(* Logix 5000 project; controller p65 vendor 1 type 14 code 85 rev 20.11; software revision 20.01; part 7 of 7 *)
(* tags used below, declared in another part *)
   Commpower : ALIAS FOR REAL00_102;
   DCMicroGridisSimulating : ALIAS FOR DINT00_23.10;
   House01current : ALIAS FOR REAL00_117;
   House01isConnected : ALIAS FOR DINT00_28.23;
   House02current : ALIAS FOR REAL00_130;
   House02isConnected : ALIAS FOR DINT00_29.13;
   House03current : ALIAS FOR REAL00_143;
   House03isConnected : ALIAS FOR DINT00_30.3;
   House04current : ALIAS FOR REAL00_156;
   House04isConnected : ALIAS FOR DINT00_30.25;
   House05current : ALIAS FOR REAL00_169;
   House05isConnected : ALIAS FOR DINT00_31.15;
   LastSolar_Power : REAL;
   Load01isConnected : ALIAS FOR DINT00_24.13;
   Load02isConnected : ALIAS FOR DINT00_25.3;
   Load03isConnected : ALIAS FOR DINT00_25.25;
   Load04isConnected : ALIAS FOR DINT00_26.15;
   Load05isConnected : ALIAS FOR DINT00_27.5;
   Loadsaccum : ALIAS FOR REAL00_30;
   Loadscurrent : ALIAS FOR REAL00_105;
   LoadscurrentHILS : ALIAS FOR plc1_local_5[0];
   LoadscurrentRaw : ALIAS FOR Local:1:I.Ch6Data;
   Loadsdifference : ALIAS FOR REAL00_106;
   LoadslastLowVoltage : ALIAS FOR DINT00_27.22;
   LoadslowVoltage : ALIAS FOR DINT00_27.23;
   LoadslowVoltageBound : ALIAS FOR REAL00_107;
   Loadspower : ALIAS FOR REAL00_108;
   Loadsrecovered : ALIAS FOR DINT00_27.24;
   LoadssampleNow : ALIAS FOR DINT00_32.3;
   LoadssampleTimer : ALIAS FOR CLTIMER00_89;
   Loadstotal : ALIAS FOR REAL00_183;
   LoadstotalTooLarge : ALIAS FOR DINT00_32.4;
   LoadstotalTooSmall : ALIAS FOR DINT00_32.5;
   Loadsvoltage : ALIAS FOR REAL00_184;
   LoadsVoltageBalanceEventFail : ALIAS FOR DINT00_32.6;
   LoadsVoltageBalanceEventSuccess : ALIAS FOR DINT00_32.7;
   LoadsVoltageBalanceFailTimer : ALIAS FOR CLTIMER00_90;
   LoadsVoltageBalanceInProcess : ALIAS FOR DINT00_32.8;
   LoadsVoltageBalanceMsg : ALIAS FOR MESSAGE00_23;
   LoadsVoltageBalanceSuccessTimer : ALIAS FOR CLTIMER00_91;
   LoadsvoltageHILS : ALIAS FOR plc1_local_5[1];
   LoadsvoltageRaw : ALIAS FOR Local:1:I.Ch8Data;
   LoadsVoltageRebalancedEventFail : ALIAS FOR DINT00_32.9;
   LoadsVoltageRebalancedEventSuccess : ALIAS FOR DINT00_32.10;
   LoadsVoltageRebalancedFailTimer : ALIAS FOR CLTIMER00_92;
   LoadsVoltageRebalancedInProcess : ALIAS FOR DINT00_32.11;
   LoadsVoltageRebalancedMsg : ALIAS FOR MESSAGE00_24;
   LoadsVoltageRebalancedSuccessTimer : ALIAS FOR CLTIMER00_93;
   Resaccum : ALIAS FOR REAL00_109;
   ResBattempt : ALIAS FOR DINT00_10;
   ResBclose : ALIAS FOR Local:3:O.Data.10;
   ResBcloseHILS : ALIAS FOR plc1_local_6[0].10;
   ResBcloseProxy : ALIAS FOR DINT00_27.25;
   ResBdeadBand : ALIAS FOR REAL00_110;
   ResBfailedToOpen : ALIAS FOR DINT00_27.26;
   ResBintForceOpen : ALIAS FOR DINT00_27.27;
   ResBintReqClose : ALIAS FOR DINT00_27.28;
   ResBisClosed : ALIAS FOR DINT00_27.29;
   ResBisOpen : ALIAS FOR DINT00_27.30;
   ResBmaxAttempts : ALIAS FOR DINT00_11;
   ResBmaxLoadCurrent : ALIAS FOR REAL00_111;
   ResBopenTimer : ALIAS FOR CLTIMER00_48;
   ResBreqClose : ALIAS FOR DINT00_27.31;
   ResBreqOpen : ALIAS FOR DINT00_28.0;
   ResBreqReset : ALIAS FOR DINT00_28.1;
   ResBretriesFailed : ALIAS FOR DINT00_28.2;
   ResBtooMuchCurrent : ALIAS FOR DINT00_28.3;
   ResBunexpectedLowCurrent : ALIAS FOR DINT00_28.4;
   RescanNotifyUser : ALIAS FOR DINT00_28.5;
   RescommandChanged : ALIAS FOR DINT00_28.6;
   RescommandChangedTimer : ALIAS FOR CLTIMER00_49;
   Rescurrent : ALIAS FOR REAL00_112;
   RescurrentHILS : ALIAS FOR plc1_local_3[6];
   RescurrentRaw : ALIAS FOR Local:1:I.Ch11Data;
   Resdeadband : ALIAS FOR REAL00_113;
   Resdifference : ALIAS FOR REAL00_114;
   ResfailedToConnect : ALIAS FOR DINT00_28.7;
   ResfailedToDisconnect : ALIAS FOR DINT00_28.8;
   ResintReqConnect : ALIAS FOR DINT00_31.23;
   ResisConnected : ALIAS FOR DINT00_31.24;
   ResisDisconnected : ALIAS FOR DINT00_31.25;
   ResnotificationTimer : ALIAS FOR CLTIMER00_85;
   ResOverCurrentConditionEventFail : ALIAS FOR DINT00_31.26;
   ResOverCurrentConditionEventSuccess : ALIAS FOR DINT00_31.27;
   ResOverCurrentConditionFailTimer : ALIAS FOR CLTIMER00_86;
   ResOverCurrentConditionInProcess : ALIAS FOR DINT00_31.28;
   ResOverCurrentConditionMsg : ALIAS FOR MESSAGE00_22;
   ResOverCurrentConditionSuccessTimer : ALIAS FOR CLTIMER00_87;
   Respower : ALIAS FOR REAL00_180;
   ResreqConnect : ALIAS FOR DINT00_31.29;
   ResreqDisconnect : ALIAS FOR DINT00_31.30;
   RessampleNow : ALIAS FOR DINT00_31.31;
   RessampleTimer : ALIAS FOR CLTIMER00_88;
   Restotal : ALIAS FOR REAL00_181;
   RestotalTooLarge : ALIAS FOR DINT00_32.0;
   RestotalTooSmall : ALIAS FOR DINT00_32.1;
   ResuserNotified : ALIAS FOR DINT00_32.2;
   Resvoltage : ALIAS FOR REAL00_182;
   ResvoltageHILS : ALIAS FOR plc1_local_3[7];
   ResvoltageRaw : ALIAS FOR Local:2:I.Ch1Data;
   Solar_Power : ALIAS FOR plc1_local_1[0];
   SolarMeasureTimer : TIMER;
   SolarPanelBclose : ALIAS FOR Local:3:O.Data.13;
   SolarPanelBcloseHILS : ALIAS FOR plc1_local_6[0].12;
   SolarPanelBcloseProxy : ALIAS FOR DINT00_32.22;
   SolarPanelBintReqClose : ALIAS FOR DINT00_32.23;
   SolarPanelBisClosed : ALIAS FOR DINT00_32.24;
   SolarPanelBisOpen : ALIAS FOR DINT00_32.25;
   SolarPanelBreqClose : ALIAS FOR DINT00_32.26;
   SolarPanelBreqOpen : ALIAS FOR DINT00_32.27;
   SolarPanelcanSupplyPower : ALIAS FOR DINT00_32.28;
   SolarPanelcommandChanged : ALIAS FOR DINT00_32.29;
   SolarPanelcommandChangedTimer : ALIAS FOR CLTIMER00_99;
   SolarPanelcurrent : ALIAS FOR REAL00_187;
   SolarPanelcurrentHILS : ALIAS FOR plc1_local_3[0];
   SolarPanelcurrentRaw : ALIAS FOR Local:1:I.Ch2Data;
   SolarPaneldeadband : ALIAS FOR REAL00_188;
   SolarPanelfailedToConnect : ALIAS FOR DINT00_32.30;
   SolarPanelfailedToDisconnect : ALIAS FOR DINT00_32.31;
   SolarPanelintReqConnect : ALIAS FOR DINT00_33.0;
   SolarPanelisConnected : ALIAS FOR DINT00_33.1;
   SolarPanelisDisconnected : ALIAS FOR DINT00_33.2;
   SolarPanelisFunctional : ALIAS FOR DINT00_33.3;
   SolarPanelpower : ALIAS FOR REAL00_190;
   SolarPanelprovidingExcessPower : ALIAS FOR DINT00_33.4;
   SolarPanelreqConnect : ALIAS FOR DINT00_33.5;
   SolarPanelreqDisconnect : ALIAS FOR DINT00_33.6;
   SolarPanelvoltage : ALIAS FOR REAL00_191;
   SolarPanelvoltageHILS : ALIAS FOR plc1_local_3[1];
   SolarPanelvoltageRaw : ALIAS FOR Local:1:I.Ch1Data;
   UsingAgents : BOOL;

PROGRAM Loads   (* main routine Loads *)
VAR
   VoltageRebalancePhase : DINT;
END_VAR

ROUTINE Loads   (* ladder *)
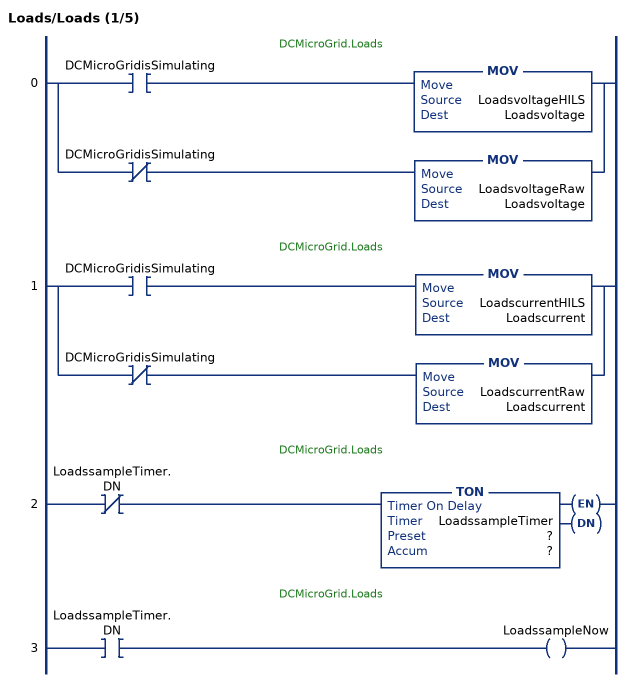
   // DCMicroGrid.Loads
   0: [XIC(DCMicroGridisSimulating) MOV(LoadsvoltageHILS,Loadsvoltage) ,XIO(DCMicroGridisSimulating) MOV(LoadsvoltageRaw,Loadsvoltage) ];
   // DCMicroGrid.Loads
   1: [XIC(DCMicroGridisSimulating) MOV(LoadscurrentHILS,Loadscurrent) ,XIO(DCMicroGridisSimulating) MOV(LoadscurrentRaw,Loadscurrent) ];
   // DCMicroGrid.Loads
   2: XIO(LoadssampleTimer.DN)TON(LoadssampleTimer,?,?);
   // DCMicroGrid.Loads
   3: XIC(LoadssampleTimer.DN)OTE(LoadssampleNow);
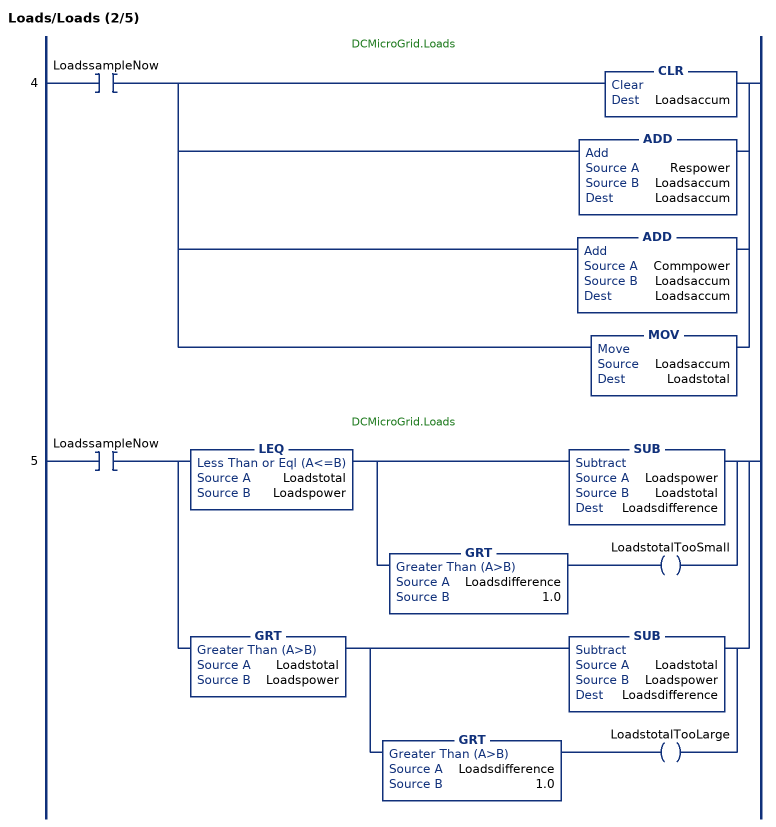
   // DCMicroGrid.Loads
   4: XIC(LoadssampleNow)[CLR(Loadsaccum) ,[ADD(Respower,Loadsaccum,Loadsaccum) ,ADD(Commpower,Loadsaccum,Loadsaccum) ] ,MOV(Loadsaccum,Loadstotal) ];
   // DCMicroGrid.Loads
   5: XIC(LoadssampleNow)[LEQ(Loadstotal,Loadspower) [SUB(Loadspower,Loadstotal,Loadsdifference) ,GRT(Loadsdifference,1.0) OTE(LoadstotalTooSmall) ] ,GRT(Loadstotal,Loadspower) [SUB(Loadstotal,Loadspower,Loadsdifference) ,GRT(Loadsdifference,1.0) OTE(LoadstotalTooLarge) ] ];
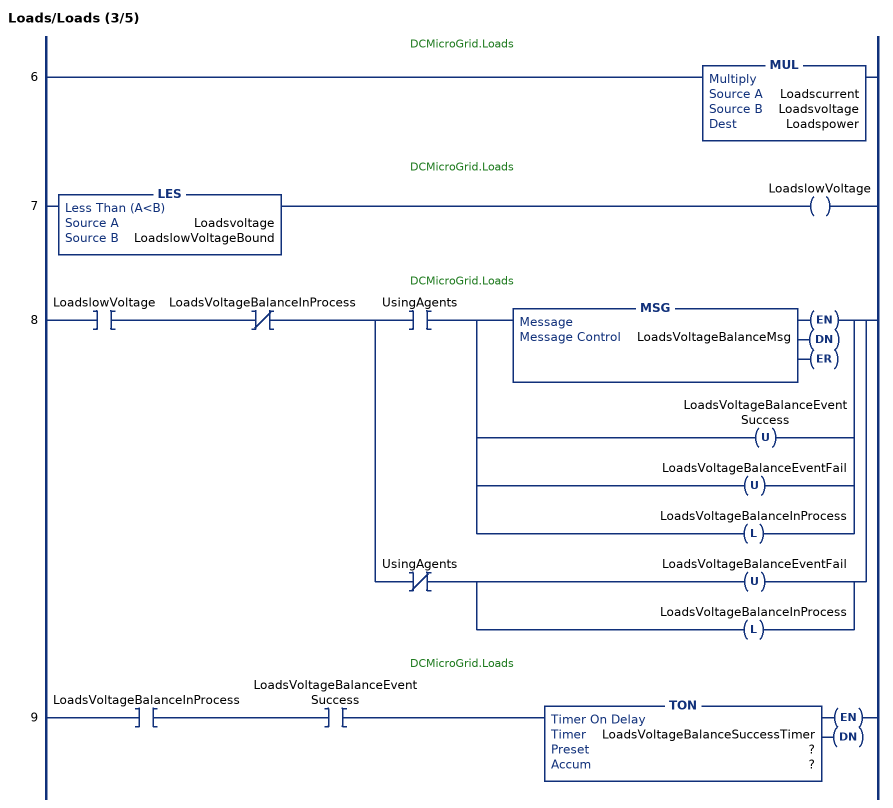
   // DCMicroGrid.Loads
   6: MUL(Loadscurrent,Loadsvoltage,Loadspower);
   // DCMicroGrid.Loads
   7: LES(Loadsvoltage,LoadslowVoltageBound)OTE(LoadslowVoltage);
   // DCMicroGrid.Loads
   8: XIC(LoadslowVoltage)XIO(LoadsVoltageBalanceInProcess)[XIC(UsingAgents) [MSG(LoadsVoltageBalanceMsg) ,OTU(LoadsVoltageBalanceEventSuccess) ,OTU(LoadsVoltageBalanceEventFail) ,OTL(LoadsVoltageBalanceInProcess) ] ,XIO(UsingAgents) [OTU(LoadsVoltageBalanceEventFail) ,OTL(LoadsVoltageBalanceInProcess) ] ];
   // DCMicroGrid.Loads
   9: XIC(LoadsVoltageBalanceInProcess)XIC(LoadsVoltageBalanceEventSuccess)TON(LoadsVoltageBalanceSuccessTimer,?,?);
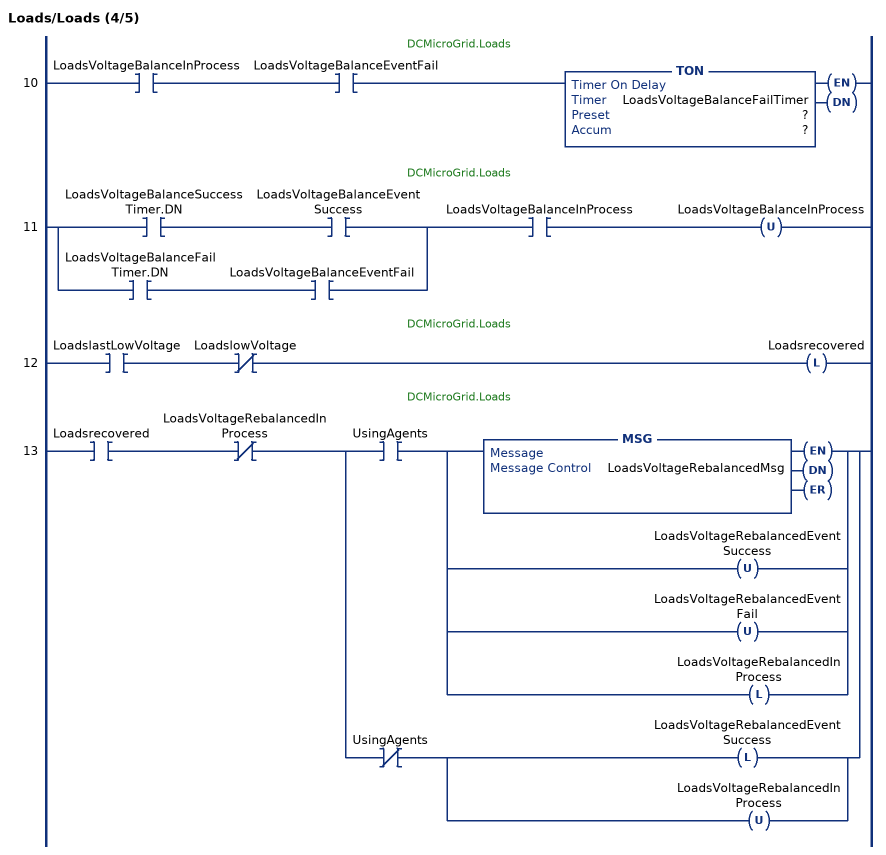
   // DCMicroGrid.Loads
   10: XIC(LoadsVoltageBalanceInProcess)XIC(LoadsVoltageBalanceEventFail)TON(LoadsVoltageBalanceFailTimer,?,?);
   // DCMicroGrid.Loads
   11: [XIC(LoadsVoltageBalanceSuccessTimer.DN) XIC(LoadsVoltageBalanceEventSuccess) ,XIC(LoadsVoltageBalanceFailTimer.DN) XIC(LoadsVoltageBalanceEventFail) ]XIC(LoadsVoltageBalanceInProcess)OTU(LoadsVoltageBalanceInProcess);
   // DCMicroGrid.Loads
   12: XIC(LoadslastLowVoltage)XIO(LoadslowVoltage)OTL(Loadsrecovered);
   // DCMicroGrid.Loads
   13: XIC(Loadsrecovered)XIO(LoadsVoltageRebalancedInProcess)[XIC(UsingAgents) [MSG(LoadsVoltageRebalancedMsg) ,OTU(LoadsVoltageRebalancedEventSuccess) ,OTU(LoadsVoltageRebalancedEventFail) ,OTL(LoadsVoltageRebalancedInProcess) ] ,XIO(UsingAgents) [OTL(LoadsVoltageRebalancedEventSuccess) ,OTU(LoadsVoltageRebalancedInProcess) ] ];
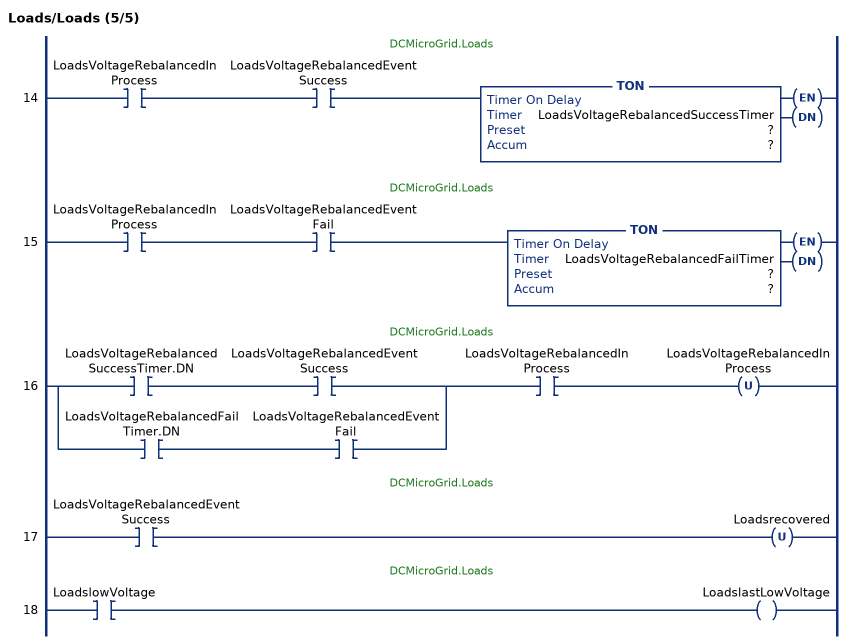
   // DCMicroGrid.Loads
   14: XIC(LoadsVoltageRebalancedInProcess)XIC(LoadsVoltageRebalancedEventSuccess)TON(LoadsVoltageRebalancedSuccessTimer,?,?);
   // DCMicroGrid.Loads
   15: XIC(LoadsVoltageRebalancedInProcess)XIC(LoadsVoltageRebalancedEventFail)TON(LoadsVoltageRebalancedFailTimer,?,?);
   // DCMicroGrid.Loads
   16: [XIC(LoadsVoltageRebalancedSuccessTimer.DN) XIC(LoadsVoltageRebalancedEventSuccess) ,XIC(LoadsVoltageRebalancedFailTimer.DN) XIC(LoadsVoltageRebalancedEventFail) ]XIC(LoadsVoltageRebalancedInProcess)OTU(LoadsVoltageRebalancedInProcess);
   // DCMicroGrid.Loads
   17: XIC(LoadsVoltageRebalancedEventSuccess)OTU(Loadsrecovered);
   // DCMicroGrid.Loads
   18: XIC(LoadslowVoltage)OTE(LoadslastLowVoltage);
END_ROUTINE
END_PROGRAM

PROGRAM Main   (* main routine PDLGeneratedControlLogic *)

ROUTINE PDLGeneratedControlLogic   (* ladder *)
END_ROUTINE
END_PROGRAM

PROGRAM Res   (* main routine Res *)

ROUTINE Res   (* ladder *)
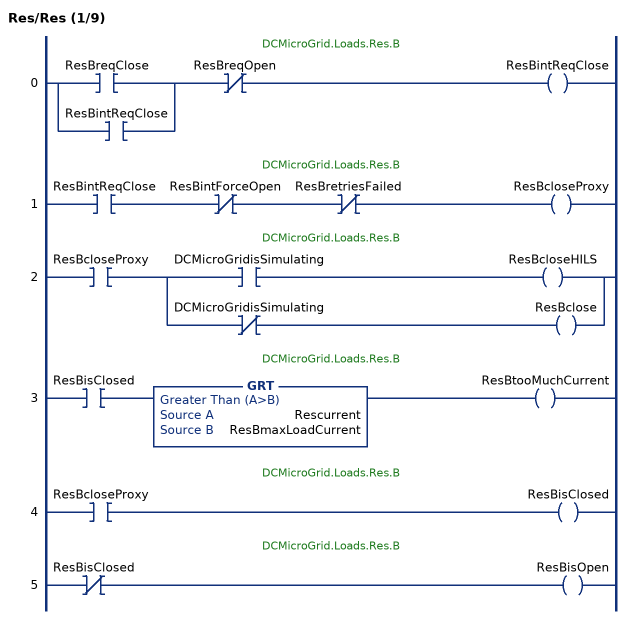
   // DCMicroGrid.Loads.Res.B
   0: [XIC(ResBreqClose) ,XIC(ResBintReqClose) ]XIO(ResBreqOpen)OTE(ResBintReqClose);
   // DCMicroGrid.Loads.Res.B
   1: XIC(ResBintReqClose)XIO(ResBintForceOpen)XIO(ResBretriesFailed)OTE(ResBcloseProxy);
   // DCMicroGrid.Loads.Res.B
   2: XIC(ResBcloseProxy)[XIC(DCMicroGridisSimulating) OTE(ResBcloseHILS) ,XIO(DCMicroGridisSimulating) OTE(ResBclose) ];
   // DCMicroGrid.Loads.Res.B
   3: XIC(ResBisClosed)GRT(Rescurrent,ResBmaxLoadCurrent)OTE(ResBtooMuchCurrent);
   // DCMicroGrid.Loads.Res.B
   4: XIC(ResBcloseProxy)OTE(ResBisClosed);
   // DCMicroGrid.Loads.Res.B
   5: XIO(ResBisClosed)OTE(ResBisOpen);
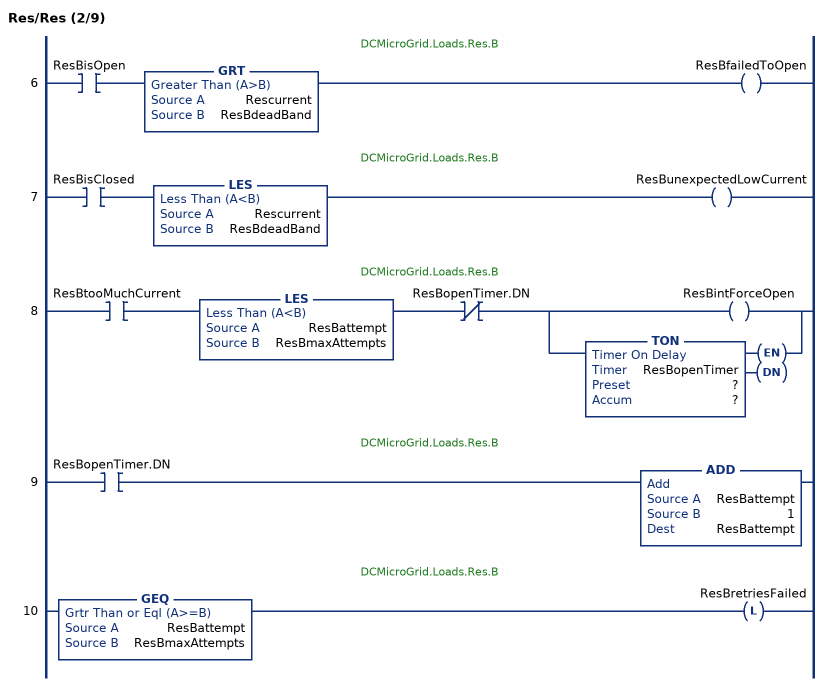
   // DCMicroGrid.Loads.Res.B
   6: XIC(ResBisOpen)GRT(Rescurrent,ResBdeadBand)OTE(ResBfailedToOpen);
   // DCMicroGrid.Loads.Res.B
   7: XIC(ResBisClosed)LES(Rescurrent,ResBdeadBand)OTE(ResBunexpectedLowCurrent);
   // DCMicroGrid.Loads.Res.B
   8: XIC(ResBtooMuchCurrent)LES(ResBattempt,ResBmaxAttempts)XIO(ResBopenTimer.DN)[OTE(ResBintForceOpen) ,TON(ResBopenTimer,?,?) ];
   // DCMicroGrid.Loads.Res.B
   9: XIC(ResBopenTimer.DN)ADD(ResBattempt,1,ResBattempt);
   // DCMicroGrid.Loads.Res.B
   10: GEQ(ResBattempt,ResBmaxAttempts)OTL(ResBretriesFailed);
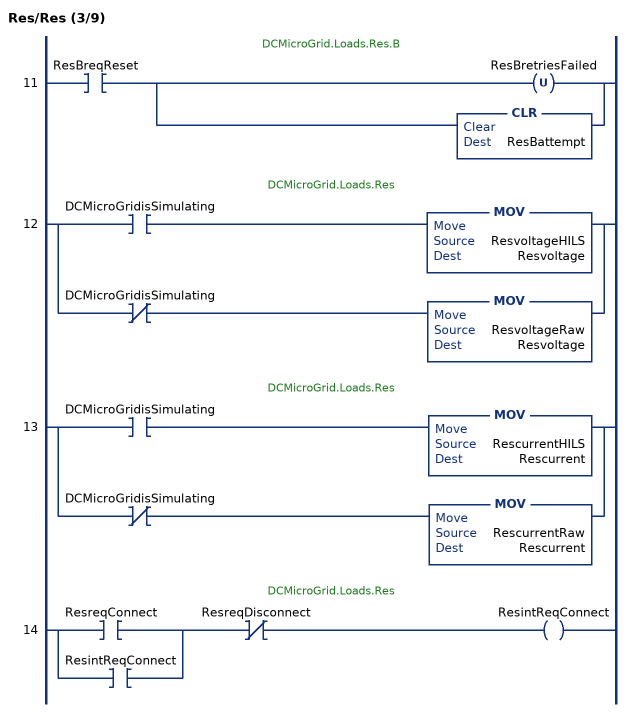
   // DCMicroGrid.Loads.Res.B
   11: XIC(ResBreqReset)[OTU(ResBretriesFailed) ,CLR(ResBattempt) ];
   // DCMicroGrid.Loads.Res
   12: [XIC(DCMicroGridisSimulating) MOV(ResvoltageHILS,Resvoltage) ,XIO(DCMicroGridisSimulating) MOV(ResvoltageRaw,Resvoltage) ];
   // DCMicroGrid.Loads.Res
   13: [XIC(DCMicroGridisSimulating) MOV(RescurrentHILS,Rescurrent) ,XIO(DCMicroGridisSimulating) MOV(RescurrentRaw,Rescurrent) ];
   // DCMicroGrid.Loads.Res
   14: [XIC(ResreqConnect) ,XIC(ResintReqConnect) ]XIO(ResreqDisconnect)OTE(ResintReqConnect);
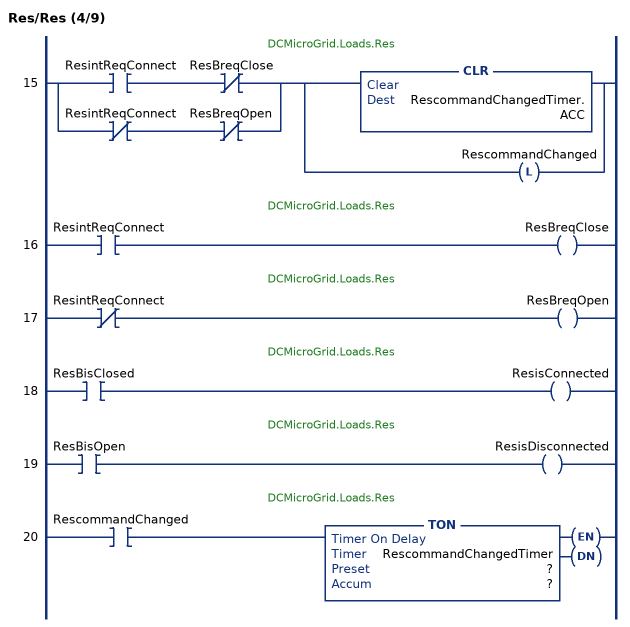
   // DCMicroGrid.Loads.Res
   15: [XIC(ResintReqConnect) XIO(ResBreqClose) ,XIO(ResintReqConnect) XIO(ResBreqOpen) ][CLR(RescommandChangedTimer.ACC) ,OTL(RescommandChanged) ];
   // DCMicroGrid.Loads.Res
   16: XIC(ResintReqConnect)OTE(ResBreqClose);
   // DCMicroGrid.Loads.Res
   17: XIO(ResintReqConnect)OTE(ResBreqOpen);
   // DCMicroGrid.Loads.Res
   18: XIC(ResBisClosed)OTE(ResisConnected);
   // DCMicroGrid.Loads.Res
   19: XIC(ResBisOpen)OTE(ResisDisconnected);
   // DCMicroGrid.Loads.Res
   20: XIC(RescommandChanged)TON(RescommandChangedTimer,?,?);
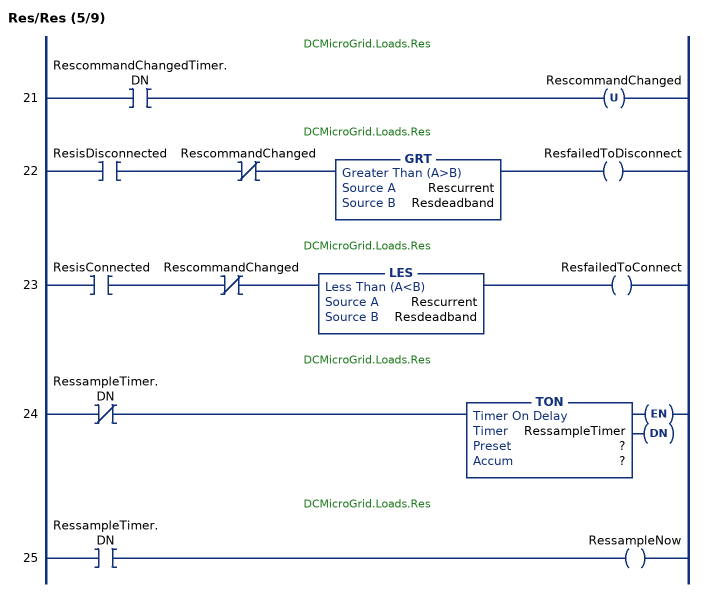
   // DCMicroGrid.Loads.Res
   21: XIC(RescommandChangedTimer.DN)OTU(RescommandChanged);
   // DCMicroGrid.Loads.Res
   22: XIC(ResisDisconnected)XIO(RescommandChanged)GRT(Rescurrent,Resdeadband)OTE(ResfailedToDisconnect);
   // DCMicroGrid.Loads.Res
   23: XIC(ResisConnected)XIO(RescommandChanged)LES(Rescurrent,Resdeadband)OTE(ResfailedToConnect);
   // DCMicroGrid.Loads.Res
   24: XIO(RessampleTimer.DN)TON(RessampleTimer,?,?);
   // DCMicroGrid.Loads.Res
   25: XIC(RessampleTimer.DN)OTE(RessampleNow);
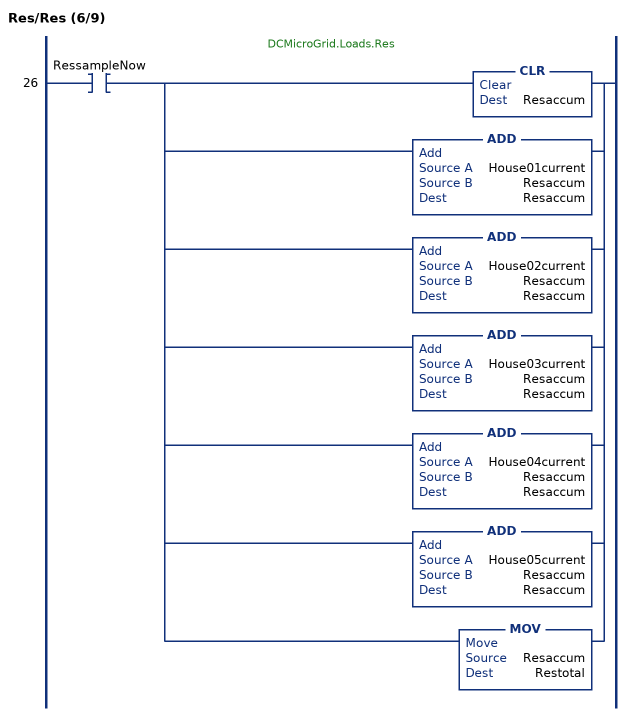
   // DCMicroGrid.Loads.Res
   26: XIC(RessampleNow)[CLR(Resaccum) ,[ADD(House01current,Resaccum,Resaccum) ,ADD(House02current,Resaccum,Resaccum) ,ADD(House03current,Resaccum,Resaccum) ,ADD(House04current,Resaccum,Resaccum) ,ADD(House05current,Resaccum,Resaccum) ] ,MOV(Resaccum,Restotal) ];
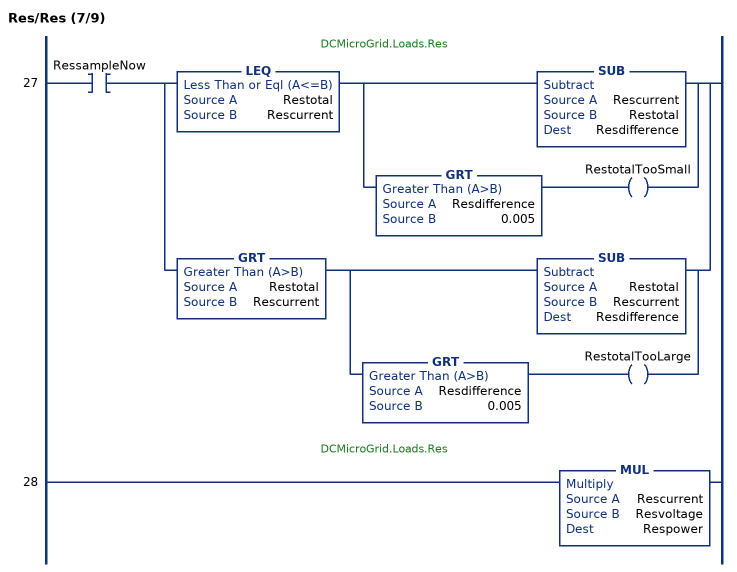
   // DCMicroGrid.Loads.Res
   27: XIC(RessampleNow)[LEQ(Restotal,Rescurrent) [SUB(Rescurrent,Restotal,Resdifference) ,GRT(Resdifference,0.005) OTE(RestotalTooSmall) ] ,GRT(Restotal,Rescurrent) [SUB(Restotal,Rescurrent,Resdifference) ,GRT(Resdifference,0.005) OTE(RestotalTooLarge) ] ];
   // DCMicroGrid.Loads.Res
   28: MUL(Rescurrent,Resvoltage,Respower);
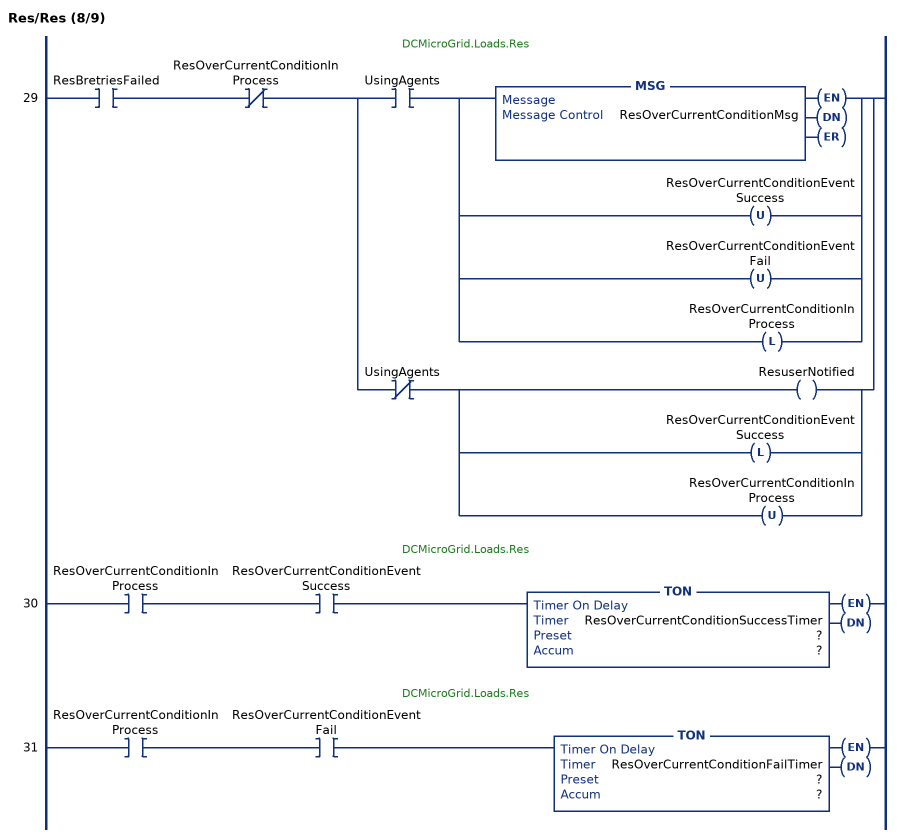
   // DCMicroGrid.Loads.Res
   29: XIC(ResBretriesFailed)XIO(ResOverCurrentConditionInProcess)[XIC(UsingAgents) [MSG(ResOverCurrentConditionMsg) ,OTU(ResOverCurrentConditionEventSuccess) ,OTU(ResOverCurrentConditionEventFail) ,OTL(ResOverCurrentConditionInProcess) ] ,XIO(UsingAgents) [OTE(ResuserNotified) ,OTL(ResOverCurrentConditionEventSuccess) ,OTU(ResOverCurrentConditionInProcess) ] ];
   // DCMicroGrid.Loads.Res
   30: XIC(ResOverCurrentConditionInProcess)XIC(ResOverCurrentConditionEventSuccess)TON(ResOverCurrentConditionSuccessTimer,?,?);
   // DCMicroGrid.Loads.Res
   31: XIC(ResOverCurrentConditionInProcess)XIC(ResOverCurrentConditionEventFail)TON(ResOverCurrentConditionFailTimer,?,?);
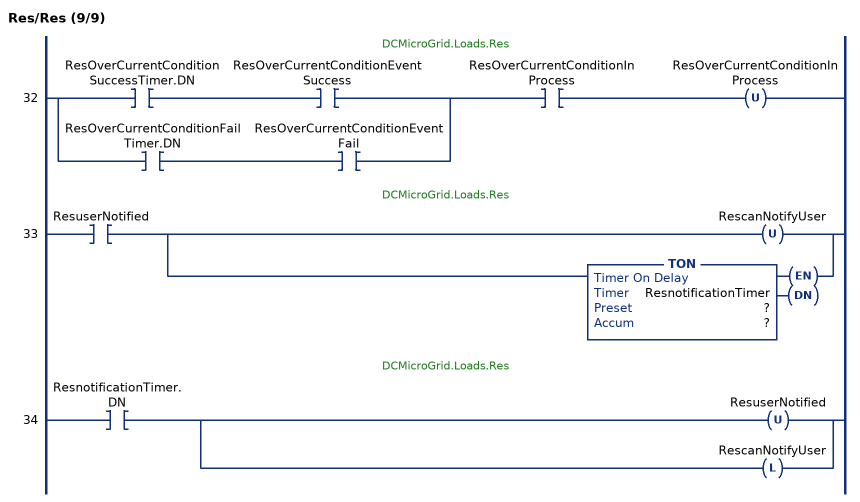
   // DCMicroGrid.Loads.Res
   32: [XIC(ResOverCurrentConditionSuccessTimer.DN) XIC(ResOverCurrentConditionEventSuccess) ,XIC(ResOverCurrentConditionFailTimer.DN) XIC(ResOverCurrentConditionEventFail) ]XIC(ResOverCurrentConditionInProcess)OTU(ResOverCurrentConditionInProcess);
   // DCMicroGrid.Loads.Res
   33: XIC(ResuserNotified)[OTU(RescanNotifyUser) ,TON(ResnotificationTimer,?,?) ];
   // DCMicroGrid.Loads.Res
   34: XIC(ResnotificationTimer.DN)[OTU(ResuserNotified) ,OTL(RescanNotifyUser) ];
END_ROUTINE
END_PROGRAM

PROGRAM SolarPanel   (* main routine SolarPanel *)

ROUTINE SolarPanel   (* ladder *)
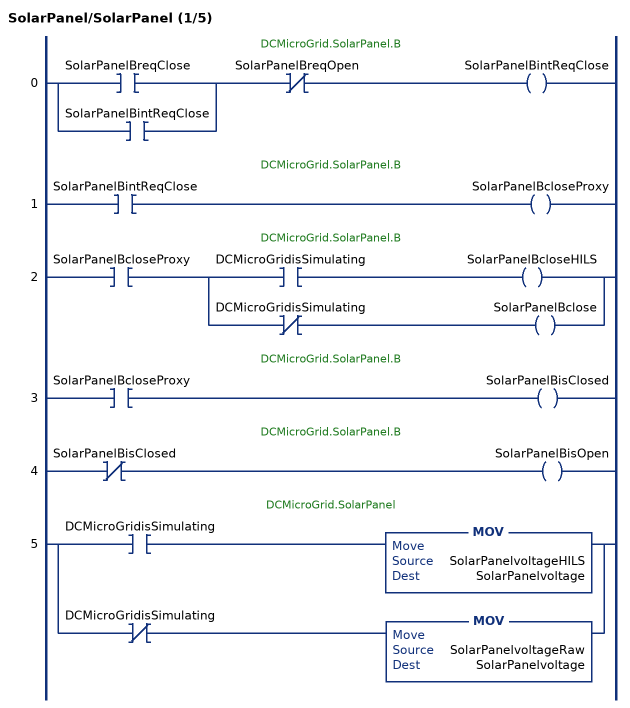
   // DCMicroGrid.SolarPanel.B
   0: [XIC(SolarPanelBreqClose) ,XIC(SolarPanelBintReqClose) ]XIO(SolarPanelBreqOpen)OTE(SolarPanelBintReqClose);
   // DCMicroGrid.SolarPanel.B
   1: XIC(SolarPanelBintReqClose)OTE(SolarPanelBcloseProxy);
   // DCMicroGrid.SolarPanel.B
   2: XIC(SolarPanelBcloseProxy)[XIC(DCMicroGridisSimulating) OTE(SolarPanelBcloseHILS) ,XIO(DCMicroGridisSimulating) OTE(SolarPanelBclose) ];
   // DCMicroGrid.SolarPanel.B
   3: XIC(SolarPanelBcloseProxy)OTE(SolarPanelBisClosed);
   // DCMicroGrid.SolarPanel.B
   4: XIO(SolarPanelBisClosed)OTE(SolarPanelBisOpen);
   // DCMicroGrid.SolarPanel
   5: [XIC(DCMicroGridisSimulating) MOV(SolarPanelvoltageHILS,SolarPanelvoltage) ,XIO(DCMicroGridisSimulating) MOV(SolarPanelvoltageRaw,SolarPanelvoltage) ];
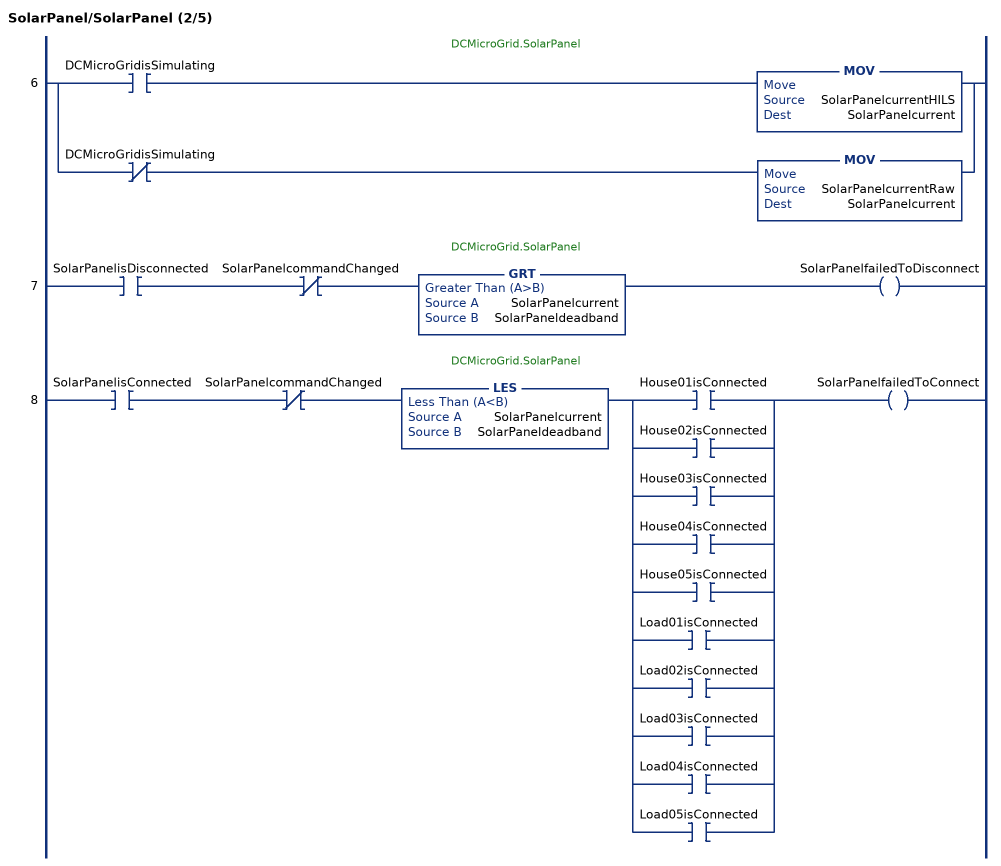
   // DCMicroGrid.SolarPanel
   6: [XIC(DCMicroGridisSimulating) MOV(SolarPanelcurrentHILS,SolarPanelcurrent) ,XIO(DCMicroGridisSimulating) MOV(SolarPanelcurrentRaw,SolarPanelcurrent) ];
   // DCMicroGrid.SolarPanel
   7: XIC(SolarPanelisDisconnected)XIO(SolarPanelcommandChanged)GRT(SolarPanelcurrent,SolarPaneldeadband)OTE(SolarPanelfailedToDisconnect);
   // DCMicroGrid.SolarPanel
   8: XIC(SolarPanelisConnected)XIO(SolarPanelcommandChanged)LES(SolarPanelcurrent,SolarPaneldeadband)[XIC(House01isConnected) ,XIC(House02isConnected) ,XIC(House03isConnected) ,XIC(House04isConnected) ,XIC(House05isConnected) ,XIC(Load01isConnected) ,XIC(Load02isConnected) ,XIC(Load03isConnected) ,XIC(Load04isConnected) ,XIC(Load05isConnected) ]OTE(SolarPanelfailedToConnect);
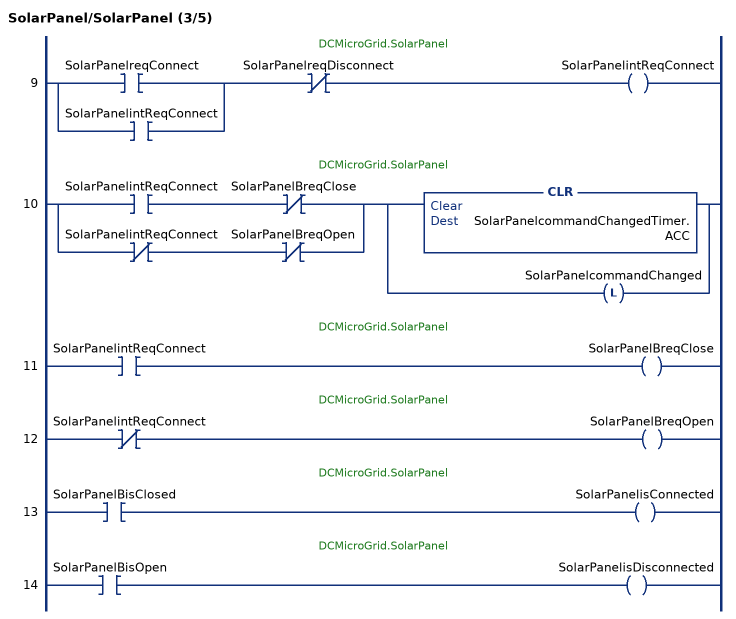
   // DCMicroGrid.SolarPanel
   9: [XIC(SolarPanelreqConnect) ,XIC(SolarPanelintReqConnect) ]XIO(SolarPanelreqDisconnect)OTE(SolarPanelintReqConnect);
   // DCMicroGrid.SolarPanel
   10: [XIC(SolarPanelintReqConnect) XIO(SolarPanelBreqClose) ,XIO(SolarPanelintReqConnect) XIO(SolarPanelBreqOpen) ][CLR(SolarPanelcommandChangedTimer.ACC) ,OTL(SolarPanelcommandChanged) ];
   // DCMicroGrid.SolarPanel
   11: XIC(SolarPanelintReqConnect)OTE(SolarPanelBreqClose);
   // DCMicroGrid.SolarPanel
   12: XIO(SolarPanelintReqConnect)OTE(SolarPanelBreqOpen);
   // DCMicroGrid.SolarPanel
   13: XIC(SolarPanelBisClosed)OTE(SolarPanelisConnected);
   // DCMicroGrid.SolarPanel
   14: XIC(SolarPanelBisOpen)OTE(SolarPanelisDisconnected);
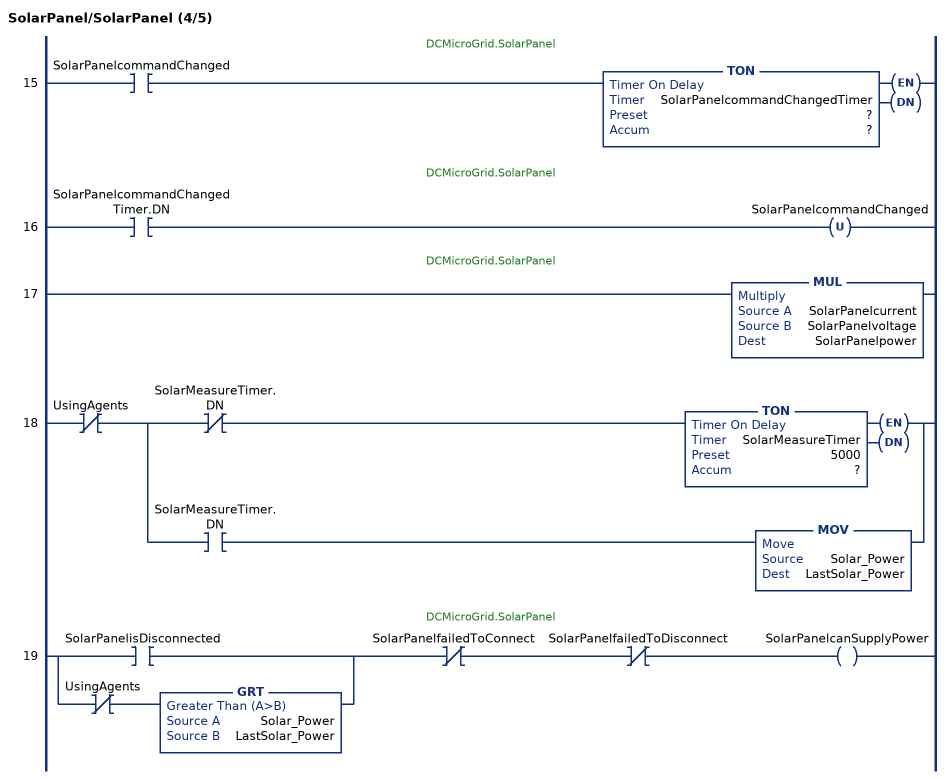
   // DCMicroGrid.SolarPanel
   15: XIC(SolarPanelcommandChanged)TON(SolarPanelcommandChangedTimer,?,?);
   // DCMicroGrid.SolarPanel
   16: XIC(SolarPanelcommandChangedTimer.DN)OTU(SolarPanelcommandChanged);
   // DCMicroGrid.SolarPanel
   17: MUL(SolarPanelcurrent,SolarPanelvoltage,SolarPanelpower);
   18: XIO(UsingAgents)[XIO(SolarMeasureTimer.DN) TON(SolarMeasureTimer,?,?) ,XIC(SolarMeasureTimer.DN) MOV(Solar_Power,LastSolar_Power) ];
   // DCMicroGrid.SolarPanel
   19: [XIC(SolarPanelisDisconnected) ,XIO(UsingAgents) GRT(Solar_Power,LastSolar_Power) ]XIO(SolarPanelfailedToConnect)XIO(SolarPanelfailedToDisconnect)OTE(SolarPanelcanSupplyPower);
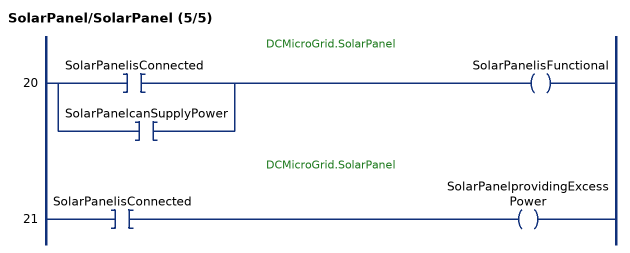
   // DCMicroGrid.SolarPanel
   20: [XIC(SolarPanelisConnected) ,XIC(SolarPanelcanSupplyPower) ]OTE(SolarPanelisFunctional);
   // DCMicroGrid.SolarPanel
   21: XIC(SolarPanelisConnected)OTE(SolarPanelprovidingExcessPower);
END_ROUTINE
END_PROGRAM
